FUNCTION_BLOCK AxisCoupledFBs
VAR_IN_OUT
	Axis					:Axis_Ref; //slave axis
	Control					:CTR_SIGNALS_INTERNAL; //master axis controls
	Output					:OUT_SIGNALS; //slave axis output
	HomeStatus				:MOTION_FB_STATUS;
END_VAR
VAR
	mcReset					:MC_Reset;
	mcPowerCoupled			:MC_Power;
	mcSetPosition			:MC_SetPosition;
	mcReadActualPosition	:MC_ReadActualPosition;
	mcReadActualVelocity	:MC_ReadActualVelocity;
	mcHome					:MC_Home;	
	mcGearIn				:MC_GearIn;
	mcGearOut				:MC_GearOut;	
	
	Zero					:LREAL:= 0;

END_VAR

mcReset(Axis := Axis, Execute := Control.Execute_C_RES); // MC_Reset
mcPowerCoupled(
    Axis := Axis,
    Enable := Control.CouplePowerEn,
    Enable_Positive := NOT Control.LimPos AND Control.CouplePowerEn,
    Enable_Negative := Control.CouplePowerEn); // MC_Power
mcSetPosition(Axis := Axis, Execute := Control.Execute_SPOS, Position := zero); // MC_SetPosition
mcReadActualPosition(Axis := Axis, Enable := Control.CouplePowerEn); // MC_ReadActualPosition
Output.PositionOut := mcReadActualPosition.Position;
mcReadActualVelocity(Axis := Axis, Enable := Control.CouplePowerEn); // MC_ReadActualVelocity
mcHome(Axis := Axis, Execute := Control.Execute_REV_HOME, bCalibrationCam := Control.LimNeg); // MC_Home
mcGearIn(Master := Axis, Slave := Control.AxisToCouple, Execute := Control.ExecuteRevCouple); // MC_GearIn
Output.VelocityOut := mcReadActualVelocity.ActualVelocity;
HomeStatus.Done := mcHome.Done;
Output.AxisCoupled := mcGearIn.InGear;
mcGearOut(Slave := Control.AxisToCouple, Execute := Control.ExecuteRevUncouple); // MC_GearOut

END_FUNCTION_BLOCK

(* stored: Version 1.1.0.1, ProductVersion 3.1.4026.12
   POU AxisCoupledFBs: Id {6466fac8-cde9-4091-b989-eab3126cec5e}, SpecialFunc None *)
